PROGRAM Alias
VAR
	i : INT := 0;
END_VAR

 //R1 : MCP**  
	
//INPUT
	//AI	
	MCP_IO.ThermalCouple[1].Temperature_raw					:= Input.R1_01_00;  //NC -
	MCP_IO.ThermalCouple[2].Temperature_raw					:= Input.R1_01_01;  
	MCP_IO.ThermalCouple[3].Temperature_raw					:= Input.R1_01_02; 
	MCP_IO.ThermalCouple[4].Temperature_raw					:= Input.R1_01_03; 

	MCP_IO.ThermalCouple[5].Temperature_raw					:= Input.R1_02_00;  //NC -
	MCP_IO.ThermalCouple[6].Temperature_raw					:= Input.R1_02_01;  
	MCP_IO.ThermalCouple[7].Temperature_raw					:= Input.R1_02_02; 
	MCP_IO.ThermalCouple[8].Temperature_raw					:= Input.R1_02_03; 
	
	MCP_IO.ThermalCouple[9].Temperature_raw					:= Input.R1_03_00;  //NC -
	MCP_IO.ThermalCouple[10].Temperature_raw				:= Input.R1_03_01;  
	MCP_IO.ThermalCouple[11].Temperature_raw				:= Input.R1_03_02; 
	MCP_IO.ThermalCouple[12].Temperature_raw				:= Input.R1_03_03; 
	
	//OUTPUT
	//AQ
	Output.R1_18_00	:= MCP_IO.ChargerSP_raw;
					
	

	
//*************************************************************************************************************

END_PROGRAM

(* stored: Version 1.1.0.1, ProductVersion 3.1.4024.11
   POU Alias: Id {ebc75665-f0df-4b03-b4d1-48515468f179}, SpecialFunc None *)
